TYPE INTERNAL ProfilerStackStruct :
STRUCT
  Hash : UDINT;
  Depth : DINT;
  StartLo : LWORD;
  StartHi : LWORD;  
  EndLo : LWORD;
  EndHi : LWORD;  
END_STRUCT
END_TYPE

(* stored: Version 1.1.0.1, ProductVersion 3.1.4024.9
   DUT ProfilerStackStruct: Id {72c79013-bc38-4419-a5a6-7aa37877a660} *)
